# EPICS substitutions: epics/db/IPOS8020.substitutions
file "./db/ecSlave.template"
{
  pattern {}
          {}
}

# No custom data yet
#file "./db/IPOS8020.template"
#{
#  pattern {}
#          {}
#}
